(* PLC project PLC1, Unknown Unnamed 1 *)
(* stored: creationDateTime 2021-02-24T14:42:08, modificationDateTime 2024-06-20T11:56:07 *)

PROGRAM PLC3
  VAR_INPUT
    level : DINT;
  END_VAR
  VAR_OUTPUT
    pump : BOOL;
  END_VAR
  VAR
    low : BOOL;
    high : BOOL;
    low_3 : DINT := 0;
    high_3 : DINT := 10;
  END_VAR

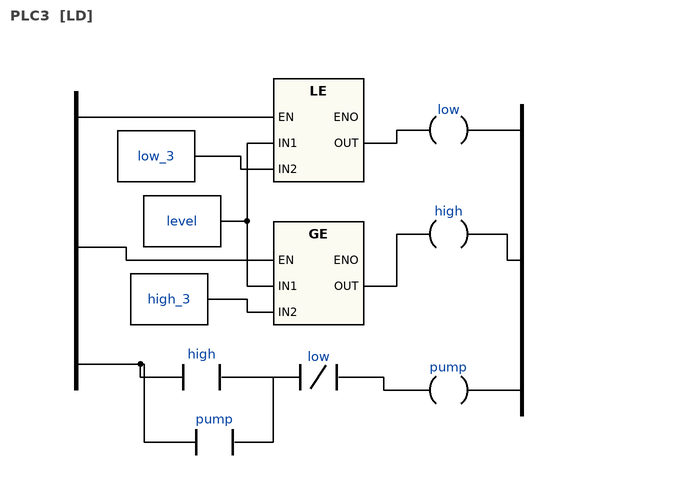
(* LD diagram, written out as Structured Text *)
high := level >= high_3;
low := level <= low_3;
pump := (high OR pump) AND NOT low;
END_PROGRAM

PROGRAM PLC2
  VAR_INPUT
    level : DINT;
  END_VAR
  VAR_OUTPUT
    request : BOOL;
  END_VAR
  VAR
    open_req : BOOL;
    close_req : BOOL;
    low_2 : DINT := 10;
    high_2 : DINT := 20;
  END_VAR

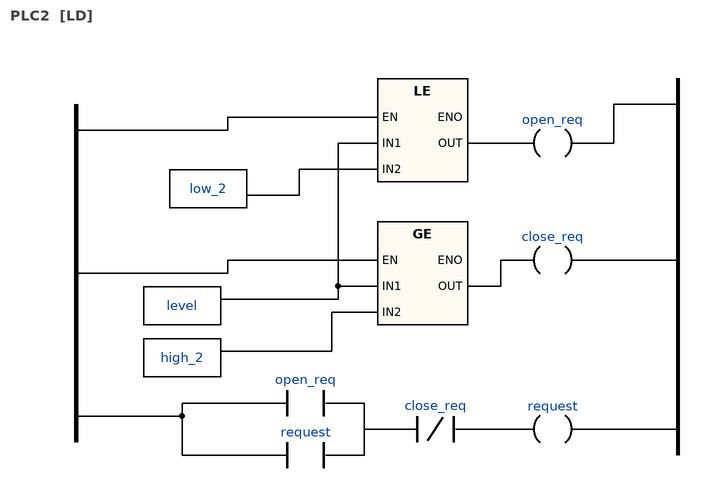
(* LD diagram, written out as Structured Text *)
close_req := level >= high_2;
open_req := level <= low_2;
request := (open_req OR request) AND NOT close_req;
END_PROGRAM

FUNCTION_BLOCK LE_0
  VAR_INPUT
    IN1 : DINT;
    IN2 : DINT;
  END_VAR
  VAR_OUTPUT
    OUT : BOOL;
  END_VAR
  VAR
    i : DINT;
    exc : __SYSTEM.ExceptionCode;
  END_VAR

            __TRY
OUT:=FALSE;
IF IN1<=IN2 then
  OUT:=TRUE;
END_IF;
IN1 : = IN2/IN1;
__CATCH(exc)
i:=IN1;
  WHILE i<4 do
    i := i * i;
  End_WHILE;
__ENDTRY;

          
END_FUNCTION_BLOCK

PROGRAM PLC1
  VAR_INPUT
    level : DINT;
    request : DINT;
  END_VAR
  VAR_OUTPUT
    pumps : BOOL;
    valve : BOOL;
  END_VAR
  VAR
    low : BOOL;
    high : BOOL;
    open_req : BOOL;
    close_req : BOOL;
    low_1 : DINT := 40;
    high_1 : DINT := 80;
    LE_00 : LE_0;
  END_VAR

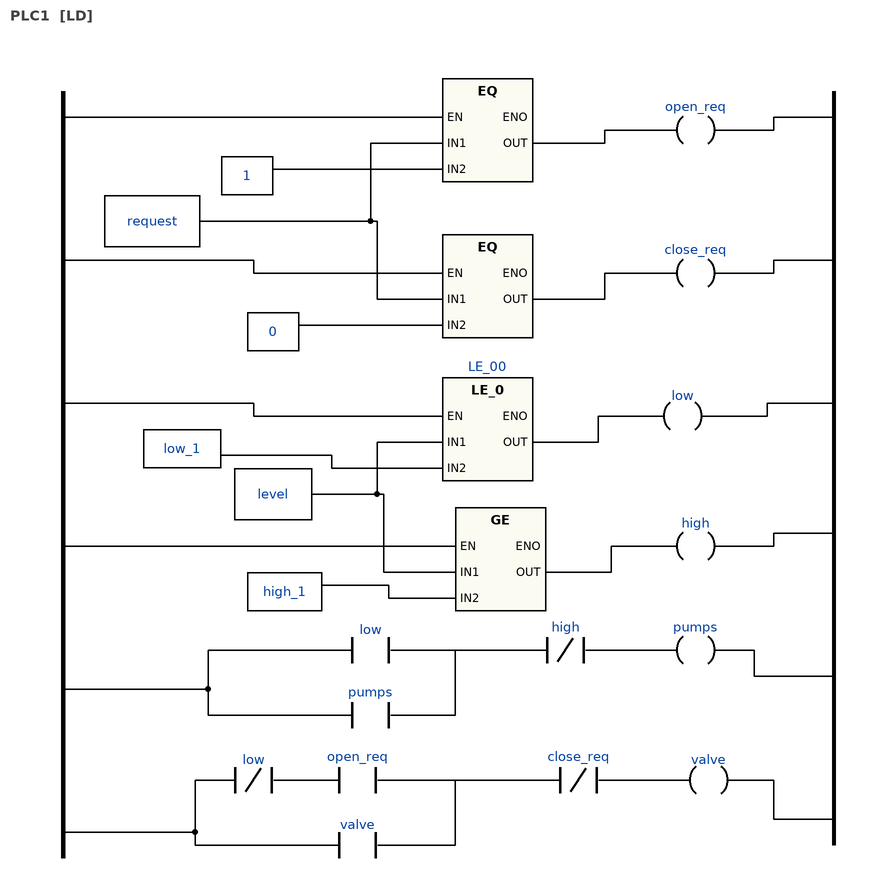
(* LD diagram, written out as Structured Text *)
open_req := request = 1;
close_req := request = 0;
pumps := (low OR pumps) AND NOT high;
valve := (NOT low AND open_req OR valve) AND NOT close_req;
LE_00(IN1 := level, IN2 := low_1);
low := LE_00.OUT;
high := level >= high_1;
END_PROGRAM

CONFIGURATION Config0
  RESOURCE Res0 ON PLC
    TASK task0(INTERVAL := T#20ms, PRIORITY := 0);
    TASK task1(INTERVAL := T#20ms, PRIORITY := 0);
    TASK task2(INTERVAL := T#20ms, PRIORITY := 0);
    PROGRAM instance0 WITH task0 : PLC1;
    PROGRAM instance1 WITH task1 : PLC2;
    PROGRAM instance2 WITH task2 : PLC3;
  END_RESOURCE
END_CONFIGURATION
